// TIA Portal V17 export
// export: Created 2024-01-30T08:49:11.3929504Z, ExportSetting WithDefaults, DisplayName Totally Integrated Automation Portal, DisplayVersion V17 Update 6, DisplayName TIA Portal Openness, DisplayVersion V17 Update 6, DisplayName TIA Portal Version Control Interface, DisplayVersion V17, DisplayName STEP 7 Professional, DisplayVersion V17 Update 6, DisplayName STEP 7 Safety, DisplayVersion V17 Update 6, DisplayName WinCC Advanced, DisplayVersion V17 Update 6
FUNCTION "FC_STL_Test" : Void   // FC1, STL
{ S7_Optimized_Access := 'TRUE' }
VERSION : 0.1
// stored: AutoNumber true, UDAEnableTagReadback false
BEGIN

NETWORK
TITLE = 
// Example how to Load Set values to ACC1 ( defined variable by T )
// L is for LOAD
// T is for TRANSFER the value from bottom ( L )

      L     125;
      T     "STL_Data".BasePos0;

      L     "STL_Data".VarBase1;
      T     "STL_Data".BasePos1;


END_FUNCTION
